FUNCTION_BLOCK IW (* Composite Function Block Type *)
  (* Standard: 61499-2 *)
  (* Version 0.0, 2016-04-07, 4DIAC-IDE, 4DIAC-Consortium *)
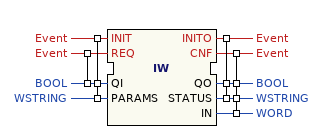
  EVENT_INPUT
    INIT WITH QI, PARAMS; (* Initialization Request *)
    REQ WITH QI; (* Normal Execution Request *)
  END_EVENT
  EVENT_OUTPUT
    INITO WITH QO, STATUS; (* Initialization Confirm *)
    CNF WITH QO, IN, STATUS; (* Execution Confirmation *)
  END_EVENT
  VAR_INPUT
    QI : BOOL; (* Input event qualifier *)
    PARAMS : WSTRING;
  END_VAR
  VAR_OUTPUT
    QO : BOOL; (* Output event qualifier *)
    STATUS : WSTRING;
    IN : WORD;
  END_VAR
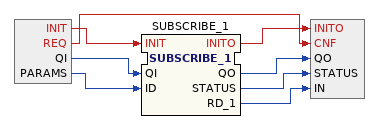
  FBS
    SUBSCRIBE_1 : SUBSCRIBE_1;
  END_FBS
  EVENT_CONNECTIONS
    INIT TO SUBSCRIBE_1.INIT;
    SUBSCRIBE_1.INITO TO INITO;
    REQ TO CNF;
  END_CONNECTIONS
  DATA_CONNECTIONS
    SUBSCRIBE_1.QO TO QO;
    SUBSCRIBE_1.STATUS TO STATUS;
    SUBSCRIBE_1.RD_1 TO IN;
    QI TO SUBSCRIBE_1.QI;
    PARAMS TO SUBSCRIBE_1.ID;
  END_CONNECTIONS
END_FUNCTION_BLOCK
